{attribute 'pack_mode' := '1'}
TYPE HomeAxis EXTENDS IncomingMessage :
STRUCT
	axisIndex: DINT; (* 1 or 2.*)
END_STRUCT
END_TYPE

(* stored: Version 1.1.0.1, ProductVersion 3.1.4022.12
   DUT HomeAxis: Id {c8f723cc-f82b-43d4-b2f5-30cd4c7ca484} *)
